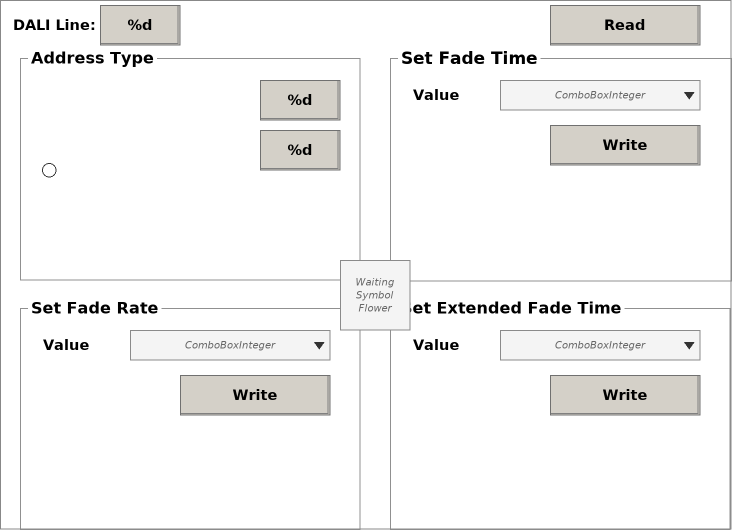
VISUALIZATION Visu_Part102SetFading  // 732x530
    GroupBox (390,50 342x231), "Set Fade Time"
        Textfield (20,30 100x30), "Value"
        ComboBoxInteger (110,30 200x30), variable: DALI_Commissioning.fbPart102SetFading.eFadeTime, text list: 'FadeTime'
        Button (160,75 150x40), "Write"
            OnMouseClick: execute { DALI_Commissioning.fbPart102SetFading.bWriteFadeTime := TRUE; }
    GroupBox (20,50 340x230), "Address Type"
        Button (240,30 80x40), "%d", text variable: DALI_Commissioning.fbPart102SetFading.nShortAddress
            OnMouseClick: write the text variable via Default, min 0, max 63, title "Insert Short Address"
        RadioButton (20,20 190x200), variable: DALI_Commissioning.fbPart102SetFading.eAddressType
            Areas[0]: Text=Short Address
            Areas[1]: Text=Group Address
            Areas[2]: Text=Broadcast
            Areas[3]: Text=Unaddressed
        Button (240,80 80x40), "%d", text variable: DALI_Commissioning.fbPart102SetFading.nGroupAddress
            OnMouseClick: write the text variable via Default, min 0, max 15, title "Insert Group Address"
    GroupBox (20,300 340x230), "Set Fade Rate"
        Textfield (20,30 100x30), "Value"
        ComboBoxInteger (110,30 200x30), variable: DALI_Commissioning.fbPart102SetFading.eFadeRate, text list: 'FadeRate'
        Button (160,75 150x40), "Write"
            OnMouseClick: execute { DALI_Commissioning.fbPart102setFading.bWriteFadeRate := TRUE; }
    GroupBox (390,300 340x230), "Set Extended Fade Time"
        Textfield (20,30 100x30), "Value"
        ComboBoxInteger (110,30 200x30), tooltip "Extended Fade Time only valid if Fade Time equals 0!", variable: DALI_Commissioning.fbPart102SetFading.eExtendedFadeTime, input disabled if: DALI_Commissioning.fbPart102SetFading.bNoFadeTime, text list: 'ExtendedFadeTime'
        Button (160,75 150x40), "Write", tooltip "Extended Fade Time only valid if Fade Time equals 0!", invisible if: DALI_Commissioning.fbPart102SetFading.bNoFadeTime, input disabled if: DALI_Commissioning.fbPart102SetFading.bNoFadeTime
            OnMouseClick: execute { DALI_Commissioning.fbPart102SetFading.bWriteExtendedFadeTime:=true; }
    Button (550,5 150x40), "Read", tooltip "Reads all Fading Parameters", invisible if: ( DALI_Commissioning.fbPart102SetFading.eAddressType >=1), input disabled if: ( DALI_Commissioning.fbPart102SetFading.eAddressType >=1)
        OnMouseClick: execute { DALI_Commissioning.fbPart102SetFading.bRead := TRUE; }
    WaitingSymbolFlower (340,260 70x70), invisible if: DALI_Commissioning.fbPart102SetFading.bHideWaitSymbol
    Group (10,5 170x40)
        Textfield (0,0 110x40), "DALI Line:"
        Button (90,0 80x40), "%d", text variable: GVL_Internal.nDALILine
            OnMouseClick: write the text variable via Default, min 1, max 10, title "Choose line"
END_VISUALIZATION

(* stored: Version 1.1.0.1
   Visu Visu_Part102SetFading: Id {f1590cf2-e94f-46a8-ad1b-b610f12980da} *)
